{attribute 'qualified_only'}
{attribute 'strict'}
TYPE E_Z1_Step :
(
	(* special steps *)
	NoStep := -32767,		// nessuno step
	Unknown := -32000,		// step sconosciuto
	
	(* Error steps *)
	NeOrError := -990,		// non abilitata o in errore
	Recovering := -980,		// azzeramento errori
		
	(* Stop *)
	Stop := 0,				// S0, stop
	
	(* Cycle *)
	Ready := 100,			// S1, pronto a ricevere pezzo
	DelayToFeeding := 120,	// S2, ritardo prima dell'avvio del nastro
	Loading := 140,			// S3, trasferimento pezzo verso Z2 
	DelayToZ2 := 160,		// S4, ritardo post sensore I5 verso Z2

	Done := 800,			// Ciclo concluso
	
	(* Stopping *)
	Stopping := 900	
);
END_TYPE
//  NoStep = '-32767'
//  Unknown = '-32000'
//  NeOrError = '-990'
//  Recovering = '-980'

(* stored: Version 1.1.0.1
   EnumerationTextList E_Z1_Step: Id {add0fde4-f244-01f4-1863-9ae6ca28f126} *)
